(* PLC project Generated.project, CODESYS CODESYS V3.5 SP19 Patch 1 *)
(* stored: creationDateTime 2026-09-14T14:47:22.379835, modificationDateTime 2026-09-14T14:47:22.379835 *)

(* values of E_ArmingBlockReason: NONE: Armement possible (au moins un axe x sens dispo); MODE_DISABLE: Mode DISABLE; POWER_CUTOFF: Coupure puissance amont (M1/M2/M3); CONTACTOR_OFF: Chaîne AU non réarmée (PowerContactorEngaged FALSE); BUCKET_BUSY: Action benne en cours (+ 1 scan de fin d'action); ALL_AXES_BLOCKED: Base OK mais aucun axe x sens sélectionné n'est disponible *)

{attribute 'qualified_only'}
{attribute 'strict'}
TYPE E_ArmingBlockReason : (NONE := 0, MODE_DISABLE := 1, POWER_CUTOFF := 2, CONTACTOR_OFF := 3, BUCKET_BUSY := 4, ALL_AXES_BLOCKED := 5);
END_TYPE
